(* IEC 61131-3 sources: com.logicals.lc3.webinar/usRTS_RPMControl_iSOC/src_FB_LIB_SAFE/Safe/Bitstring, 4 files *)

(* ---- wAND_SAFEBOOL.iecst ---- *)
NAMESPACE logicals.web.standard.safe
NAMESPACE bitstring

/*
 * Function block wrapper for IEC 61131-3 AND<br>
 * IN1 =  1st value (SAFEBOOL)<br>
 * IN2 =  2nd value (SAFEBOOL)<br>
 * OUT = IN1 AND IN2 (SAFEBOOL)<br>
 */
FUNCTION_BLOCK wAND_SAFEBOOL
	{ vNameAlignment:="center"; altName:="&"; bgColor:="Gold"; width:=40; hideIONames; }
	VAR_INPUT
		IN1 : SAFEBOOL;
		IN2 : SAFEBOOL;
	END_VAR
	VAR_OUTPUT
		OUT: SAFEBOOL;
	END_VAR

	IF (AND(IN1:=IN1<>SAFEBOOL_Constant#SAFEFALSE, IN2:=IN2<>SAFEBOOL_Constant#SAFEFALSE, ENO=>ENO) <> FALSE)
	THEN
		OUT := SAFEBOOL_Constant#SAFETRUE;
	ELSE
		OUT := SAFEBOOL_Constant#SAFEFALSE;
	END_IF;
	ENO := ENO AND CheckSAFEBOOL(IN1) AND CheckSAFEBOOL(IN2);
END_FUNCTION_BLOCK

END_NAMESPACE
END_NAMESPACE

(* ---- wAND_SAFEBOOL_BOOL.iecst ---- *)
NAMESPACE logicals.web.standard.safe
NAMESPACE bitstring

/*
 * Function block wrapper for IEC 61131-3 AND<br>
 * IN1 =  1st value (SAFEBOOL)<br>
 * IN2 =  2nd value (BOOL)<br>
 * OUT = IN1 AND IN2 (SAFEBOOL)<br>
 */
FUNCTION_BLOCK wAND_SAFEBOOL_BOOL
	{ vNameAlignment:="center"; altName:="&"; bgColor:="Gold"; width:=40; hideIONames; }
	VAR_INPUT
		IN1 : SAFEBOOL;
		IN2 : BOOL;
	END_VAR
	VAR_OUTPUT
		OUT: SAFEBOOL;
	END_VAR

	IF (AND(IN1:=IN1<>SAFEBOOL_Constant#SAFEFALSE, IN2:=IN2<>FALSE, ENO=>ENO) <> FALSE)
	THEN
		OUT := SAFEBOOL_Constant#SAFETRUE;
	ELSE
		OUT := SAFEBOOL_Constant#SAFEFALSE;
	END_IF;
	ENO := ENO AND CheckSAFEBOOL(IN1);
END_FUNCTION_BLOCK

END_NAMESPACE
END_NAMESPACE

(* ---- wNOT_SAFEBOOL.iecst ---- *)
NAMESPACE logicals.web.standard.safe
NAMESPACE bitstring

/*
 * Function block wrapper for IEC 61131-3 NOT<br>
 * IN = input (SAFEBOOL)<br>
 * OUT = !IN (SAFEBOOL)<br>
 */
FUNCTION_BLOCK wNOT_SAFEBOOL
	{ vNameAlignment:="center"; altName:="NOT"; bgColor:="Gold"; width:=60; hideIONames; }
	VAR_INPUT
		IN : SAFEBOOL;
	END_VAR
	VAR_OUTPUT
		OUT: SAFEBOOL;
	END_VAR

	IF (NOT(IN:=IN<>SAFEBOOL_Constant#SAFEFALSE, ENO=>ENO) <> FALSE)
	THEN
		OUT := SAFEBOOL_Constant#SAFETRUE;
	ELSE
		OUT := SAFEBOOL_Constant#SAFEFALSE;
	END_IF;
	ENO := ENO AND CheckSAFEBOOL(IN);
END_FUNCTION_BLOCK

END_NAMESPACE
END_NAMESPACE

(* ---- wOR_SAFEBOOL.iecst ---- *)
NAMESPACE logicals.web.standard.safe
NAMESPACE bitstring

/*
 * Function block wrapper for IEC 61131-3 OR<br>
 * IN1 =  1st value (SAFEBOOL)<br>
 * IN2 =  2nd value (SAFEBOOL)<br>
 * OUT = IN1 OR IN2 (SAFEBOOL)<br>
 */
FUNCTION_BLOCK wOR_SAFEBOOL
	{ vNameAlignment:="center"; altName:=">=1"; bgColor:="Gold"; width:=40; hideIONames; }
	VAR_INPUT
		IN1 : SAFEBOOL;
		IN2 : SAFEBOOL;
	END_VAR
	VAR_OUTPUT
		OUT: SAFEBOOL;
	END_VAR

	IF (OR(IN1:=IN1<>SAFEBOOL_Constant#SAFEFALSE, IN2:=IN2<>SAFEBOOL_Constant#SAFEFALSE, ENO=>ENO) <> FALSE)
	THEN
		OUT := SAFEBOOL_Constant#SAFETRUE;
	ELSE
		OUT := SAFEBOOL_Constant#SAFEFALSE;
	END_IF;
	ENO := ENO AND CheckSAFEBOOL(IN1) AND CheckSAFEBOOL(IN2);
END_FUNCTION_BLOCK

END_NAMESPACE
END_NAMESPACE
